(* PLC project faults, TNI-Software ControlBuild 4.00.17 *)
(* stored: creationDateTime 2005-06-20T11:52:52-01:00 *)

FUNCTION_BLOCK cmd_equipment_library.faults
  VAR_INPUT  (* CB.group=Orders CB.kind=inputVars *)
    forwardCmd : BOOL := false;  (* CB.mnemonicPatternPropertyName=<SY>_CMDAV_<NU> CB.libelle=Forward command *)
    backwardCmd : BOOL := false;  (* CB.mnemonicPatternPropertyName=<SY>_CMDAR_<NU> CB.libelle=Backward command *)
    highSpeedCmd : BOOL := false;  (* CB.mnemonicPatternPropertyName=hSCmd<SY><NU> CB.libelle=High speed command *)
    lowSpeedCmd : BOOL := false;  (* CB.mnemonicPatternPropertyName=lSCmd<SY><NU> CB.libelle=Low speed command *)
  END_VAR
  VAR_INPUT  (* CB.group=FeedBacks CB.kind=inputVars *)
    thermalFB : BOOL := false;  (* CB.mnemonicPatternPropertyName=<SY>_THER_<NU> CB.libelle=Feedback of the thermal protection of the engine *)
    forwardFB : BOOL := false;  (* CB.mnemonicPatternPropertyName=<SY>_RCAV_<NU> CB.libelle=Forward feedback *)
    backwardFB : BOOL := false;  (* CB.mnemonicPatternPropertyName=<SY>_RCAR_<NU> CB.libelle=Backward feedback *)
    highSpeedFB : BOOL := false;  (* CB.mnemonicPatternPropertyName=<SY>_RCGV_<NU> CB.libelle=High speed feedback *)
    lowSpeedFB : BOOL := false;  (* CB.mnemonicPatternPropertyName=<SY>_RCPV_<NU> CB.libelle=Low speed feedback *)
  END_VAR
  VAR_INPUT  (* CB.kind=inputVars *)
    acknowledgePB : BOOL := false;  (* CB.mnemonicPatternPropertyName=<SY>BPACQ<NU> CB.libelle=Acknowledgement pushbutton *)
  END_VAR
  VAR_OUTPUT  (* CB.kind=outputVars *)
    generalFault : BOOL := false;  (* CB.mnemonicPatternPropertyName=grlFlt<SY><NU> CB.libelle=General fault of the engine *)
  END_VAR
  VAR CONSTANT  (* CB.kind=parameterVars *)
    preset : DINT := 2;  (* CB.mnemonicPatternPropertyName=preset<SY><NU> *)
  END_VAR
  VAR  (* CB.group=Faults CB.kind=overControlVars *)
    thermalFault : BOOL := false;  (* CB.mnemonicPatternPropertyName=thermalFlt<SY><NU> CB.libelle=Thermal (electric) fault *)
    forwardFBFault : BOOL := false;  (* CB.mnemonicPatternPropertyName=fwdFBFlt<SY><NU> CB.libelle=Fault of the forward feedback *)
    backwardFBFault : BOOL := false;  (* CB.mnemonicPatternPropertyName=bwdFBFlt<SY><NU> CB.libelle=Fault of the backward feedback *)
  END_VAR

(* LD diagram, written out as Structured Text *)
1:
IF acknowledgePB THEN thermalFault := FALSE; END_IF;
IF acknowledgePB THEN forwardFBFault := FALSE; END_IF;
IF acknowledgePB THEN backwardFBFault := FALSE; END_IF;
IF acknowledgePB THEN generalFault := FALSE; END_IF;
2:
ton_sec_1(IN := forwardCmd AND (lowSpeedCmd OR highSpeedCmd), PT := preset);
IF ton_sec_1.Q AND (NOT forwardFB OR highSpeedCmd AND NOT highSpeedFB OR lowSpeedCmd AND NOT lowSpeedFB) THEN forwardFBFault := TRUE; END_IF;
ton_sec_2(IN := backwardCmd AND (highSpeedCmd OR lowSpeedCmd), PT := preset);
IF ton_sec_2.Q AND (NOT backwardFB OR lowSpeedCmd AND NOT lowSpeedFB OR highSpeedCmd AND NOT highSpeedFB) THEN backwardFBFault := TRUE; END_IF;
3:
ton_sec_3(IN := NOT thermalFB, PT := preset);
IF ton_sec_3.Q THEN thermalFault := TRUE; END_IF;
4:
IF thermalFault OR forwardFBFault OR backwardFBFault THEN generalFault := TRUE; END_IF;
END_FUNCTION_BLOCK
